(* Logix 5000 project; controller SX_V040001_C001 vendor 1 type 14 code 77 rev 16.23; software revision 16.04; part 25 of 35 *)
(* tags used below, declared in another part *)
   ALL_KINDS : INT[90];
   DRIVE : INT[32];
   Drive_diff_rpm_real : REAL;
   DRIVE_INTERVAL : INT[8];
   Drive_set_prop_rpm_real : REAL;
   EMPTYING : INT[18];
   G_DInput : DINT[3];
   loading : INT[19];
   METERING : INT[44];
   PARAMETER : INT[501];
(* MainProgram, continued *)

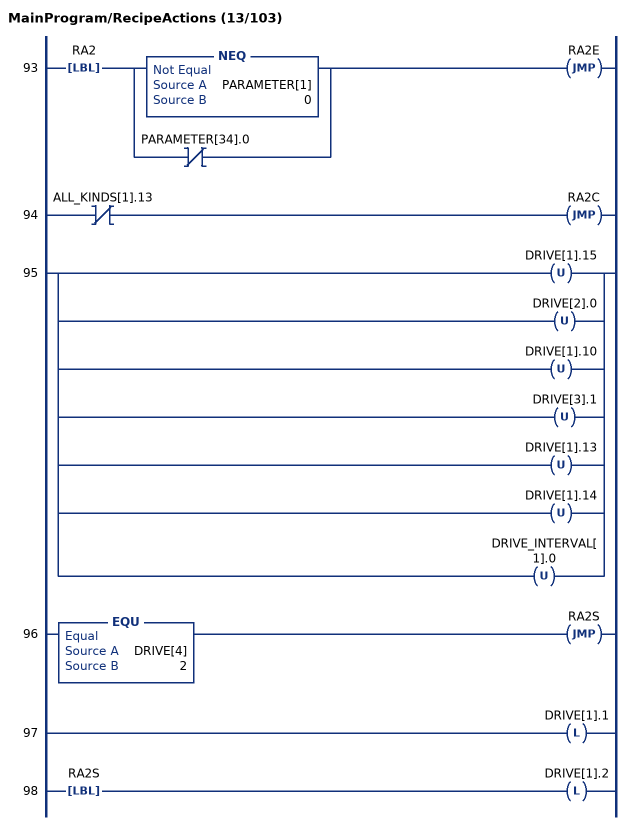
   [picture p547: MainProgram/RecipeActions rungs 93-98]
   93: LBL(RA2)[NEQ(PARAMETER[1],0) ,XIO(PARAMETER[34].0) ]JMP(RA2E);
   94: XIO(ALL_KINDS[1].13)JMP(RA2C);
   95: [OTU(DRIVE[1].15) ,OTU(DRIVE[2].0) ,OTU(DRIVE[1].10) ,OTU(DRIVE[3].1) ,OTU(DRIVE[1].13) ,OTU(DRIVE[1].14) ,OTU(DRIVE_INTERVAL[1].0) ];
   96: EQU(DRIVE[4],2)JMP(RA2S);
   97: OTL(DRIVE[1].1);
   98: LBL(RA2S)OTL(DRIVE[1].2);
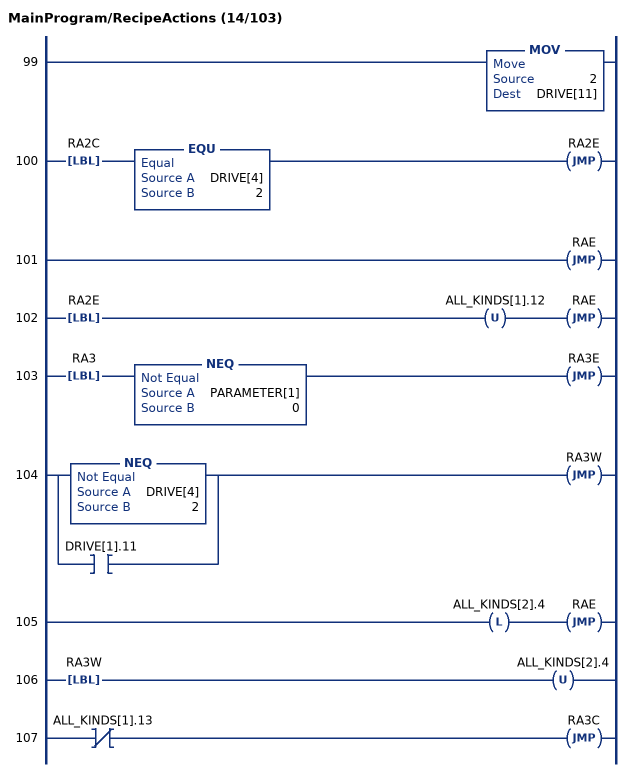
   99: MOV(2,DRIVE[11]);
   100: LBL(RA2C)EQU(DRIVE[4],2)JMP(RA2E);
   101: JMP(RAE);
   102: LBL(RA2E)OTU(ALL_KINDS[1].12)JMP(RAE);
   103: LBL(RA3)NEQ(PARAMETER[1],0)JMP(RA3E);
   104: [NEQ(DRIVE[4],2) ,XIC(DRIVE[1].11) ]JMP(RA3W);
   105: OTL(ALL_KINDS[2].4)JMP(RAE);
   106: LBL(RA3W)OTU(ALL_KINDS[2].4);
   107: XIO(ALL_KINDS[1].13)JMP(RA3C);
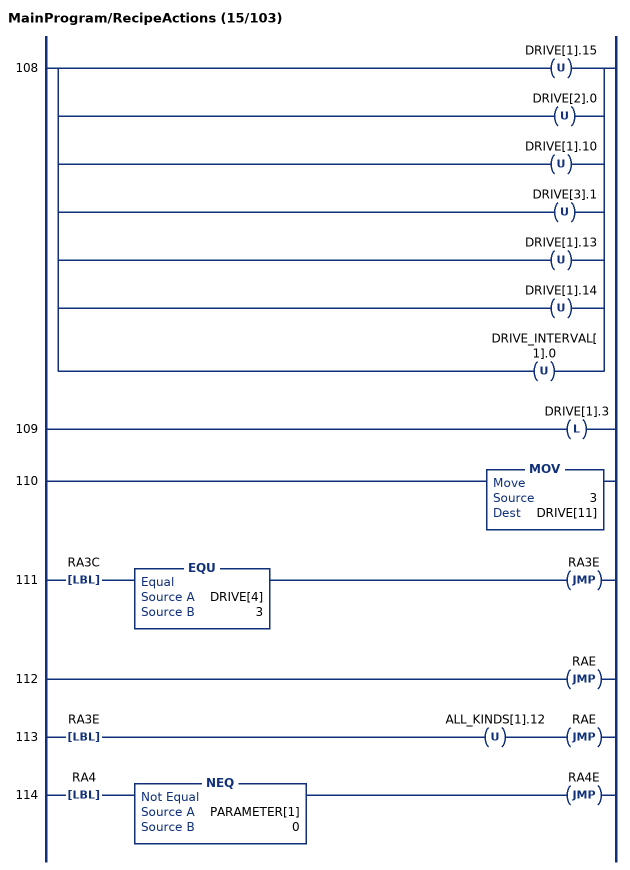
   108: [OTU(DRIVE[1].15) ,OTU(DRIVE[2].0) ,OTU(DRIVE[1].10) ,OTU(DRIVE[3].1) ,OTU(DRIVE[1].13) ,OTU(DRIVE[1].14) ,OTU(DRIVE_INTERVAL[1].0) ];
   109: OTL(DRIVE[1].3);
   110: MOV(3,DRIVE[11]);
   111: LBL(RA3C)EQU(DRIVE[4],3)JMP(RA3E);
   112: JMP(RAE);
   113: LBL(RA3E)OTU(ALL_KINDS[1].12)JMP(RAE);
   114: LBL(RA4)NEQ(PARAMETER[1],0)JMP(RA4E);
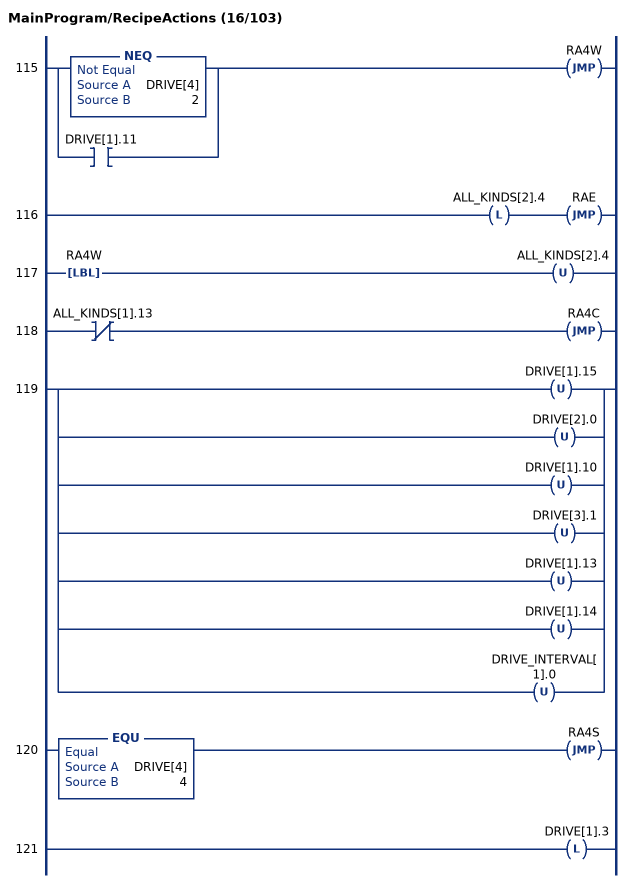
   115: [NEQ(DRIVE[4],2) ,XIC(DRIVE[1].11) ]JMP(RA4W);
   116: OTL(ALL_KINDS[2].4)JMP(RAE);
   117: LBL(RA4W)OTU(ALL_KINDS[2].4);
   118: XIO(ALL_KINDS[1].13)JMP(RA4C);
   119: [OTU(DRIVE[1].15) ,OTU(DRIVE[2].0) ,OTU(DRIVE[1].10) ,OTU(DRIVE[3].1) ,OTU(DRIVE[1].13) ,OTU(DRIVE[1].14) ,OTU(DRIVE_INTERVAL[1].0) ];
   120: EQU(DRIVE[4],4)JMP(RA4S);
   121: OTL(DRIVE[1].3);
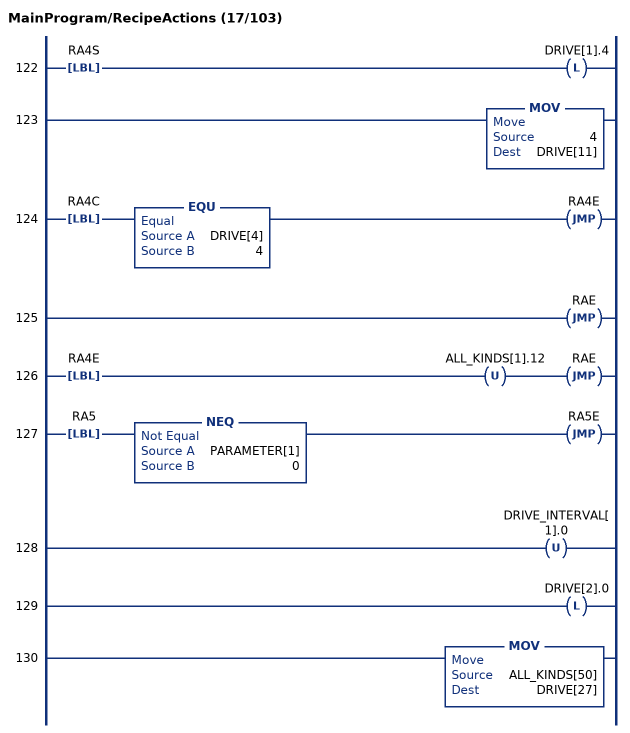
   122: LBL(RA4S)OTL(DRIVE[1].4);
   123: MOV(4,DRIVE[11]);
   124: LBL(RA4C)EQU(DRIVE[4],4)JMP(RA4E);
   125: JMP(RAE);
   126: LBL(RA4E)OTU(ALL_KINDS[1].12)JMP(RAE);
   127: LBL(RA5)NEQ(PARAMETER[1],0)JMP(RA5E);
   128: OTU(DRIVE_INTERVAL[1].0);
   129: OTL(DRIVE[2].0);
   130: MOV(ALL_KINDS[50],DRIVE[27]);
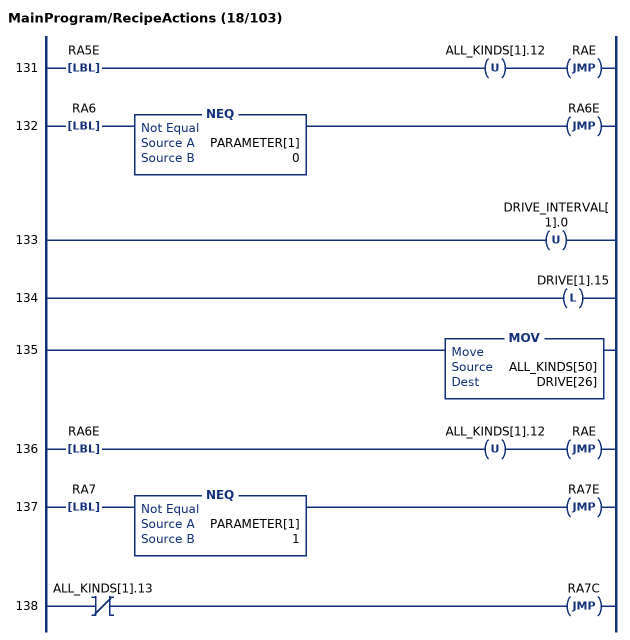
   131: LBL(RA5E)OTU(ALL_KINDS[1].12)JMP(RAE);
   132: LBL(RA6)NEQ(PARAMETER[1],0)JMP(RA6E);
   133: OTU(DRIVE_INTERVAL[1].0);
   134: OTL(DRIVE[1].15);
   135: MOV(ALL_KINDS[50],DRIVE[26]);
   136: LBL(RA6E)OTU(ALL_KINDS[1].12)JMP(RAE);
   137: LBL(RA7)NEQ(PARAMETER[1],1)JMP(RA7E);
   138: XIO(ALL_KINDS[1].13)JMP(RA7C);
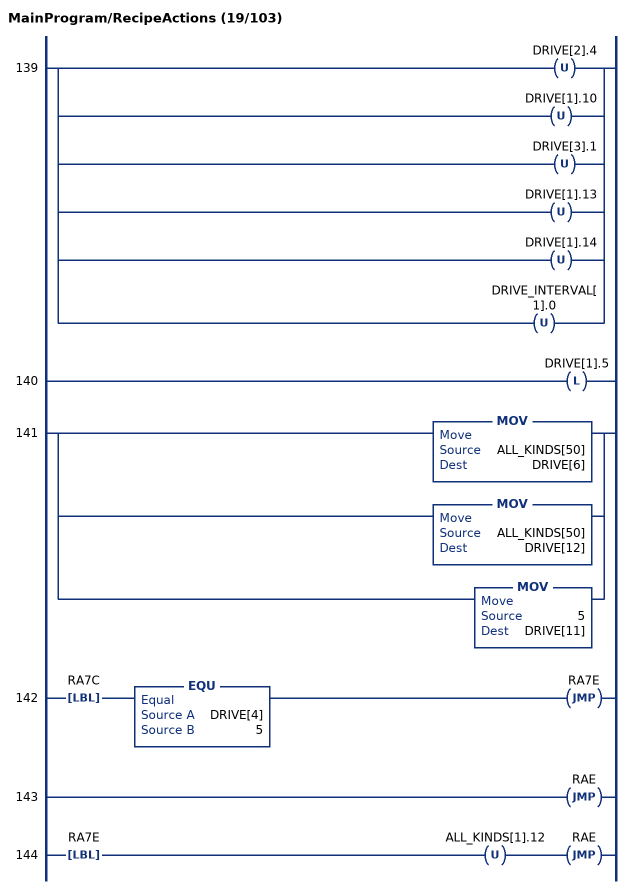
   139: [OTU(DRIVE[2].4) ,OTU(DRIVE[1].10) ,OTU(DRIVE[3].1) ,OTU(DRIVE[1].13) ,OTU(DRIVE[1].14) ,OTU(DRIVE_INTERVAL[1].0) ];
   140: OTL(DRIVE[1].5);
   141: [MOV(ALL_KINDS[50],DRIVE[6]) ,MOV(ALL_KINDS[50],DRIVE[12]) ,MOV(5,DRIVE[11]) ];
   142: LBL(RA7C)EQU(DRIVE[4],5)JMP(RA7E);
   143: JMP(RAE);
   144: LBL(RA7E)OTU(ALL_KINDS[1].12)JMP(RAE);
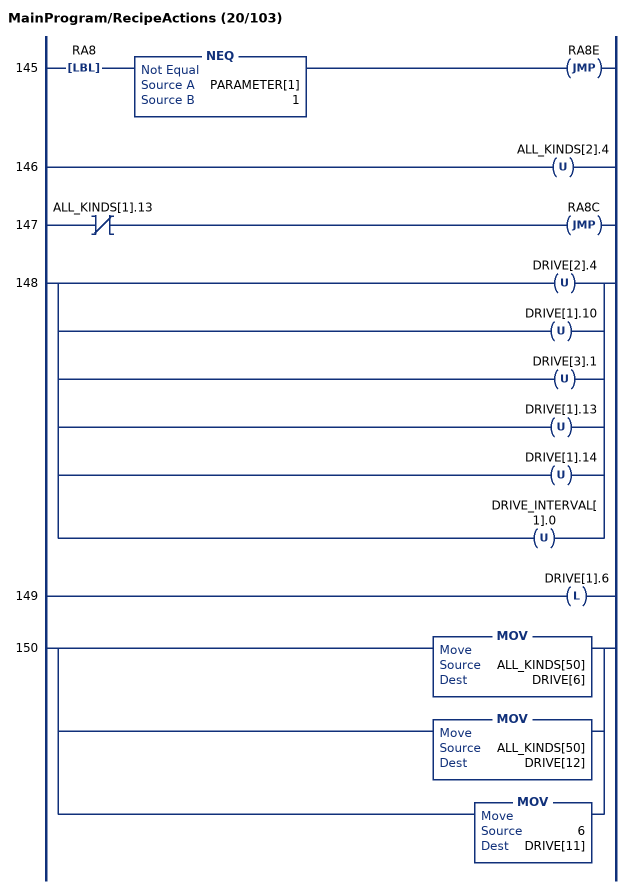
   145: LBL(RA8)NEQ(PARAMETER[1],1)JMP(RA8E);
   146: OTU(ALL_KINDS[2].4);
   147: XIO(ALL_KINDS[1].13)JMP(RA8C);
   148: [OTU(DRIVE[2].4) ,OTU(DRIVE[1].10) ,OTU(DRIVE[3].1) ,OTU(DRIVE[1].13) ,OTU(DRIVE[1].14) ,OTU(DRIVE_INTERVAL[1].0) ];
   149: OTL(DRIVE[1].6);
   150: [MOV(ALL_KINDS[50],DRIVE[6]) ,MOV(ALL_KINDS[50],DRIVE[12]) ,MOV(6,DRIVE[11]) ];
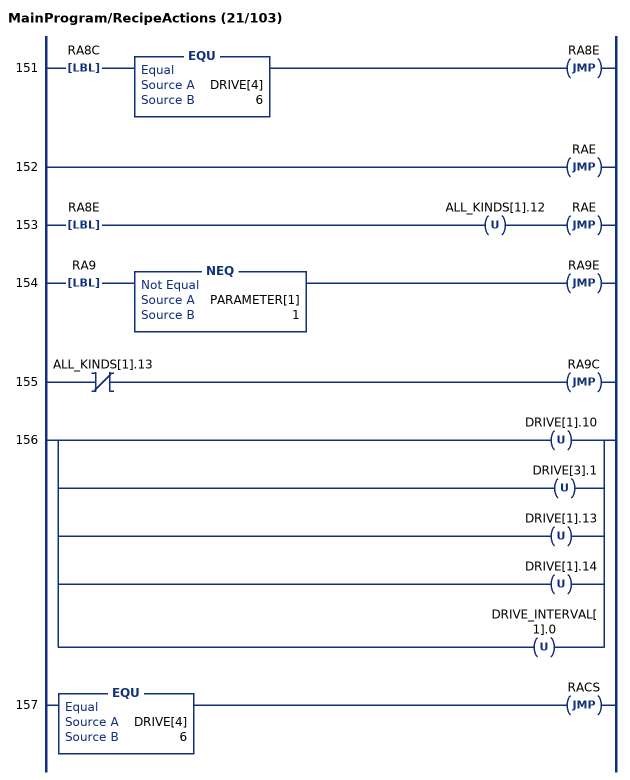
   151: LBL(RA8C)EQU(DRIVE[4],6)JMP(RA8E);
   152: JMP(RAE);
   153: LBL(RA8E)OTU(ALL_KINDS[1].12)JMP(RAE);
   154: LBL(RA9)NEQ(PARAMETER[1],1)JMP(RA9E);
   155: XIO(ALL_KINDS[1].13)JMP(RA9C);
   156: [OTU(DRIVE[1].10) ,OTU(DRIVE[3].1) ,OTU(DRIVE[1].13) ,OTU(DRIVE[1].14) ,OTU(DRIVE_INTERVAL[1].0) ];
   157: EQU(DRIVE[4],6)JMP(RACS);
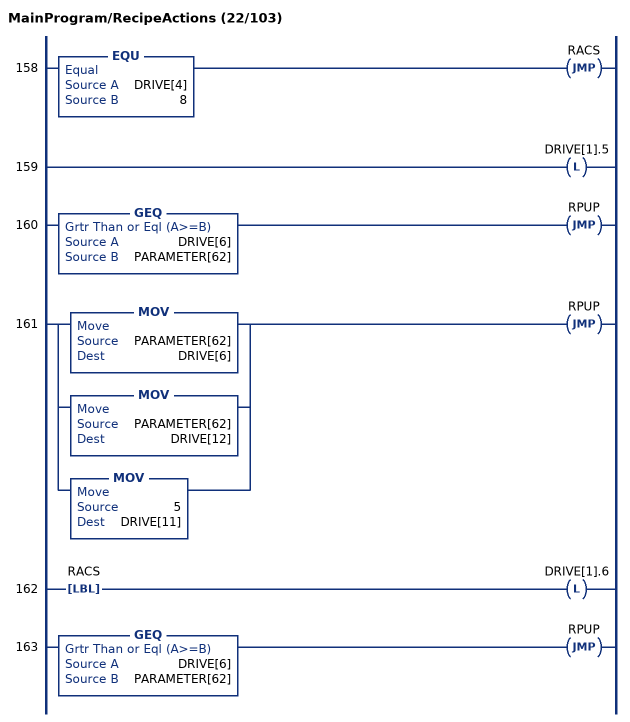
   158: EQU(DRIVE[4],8)JMP(RACS);
   159: OTL(DRIVE[1].5);
   160: GEQ(DRIVE[6],PARAMETER[62])JMP(RPUP);
   161: [MOV(PARAMETER[62],DRIVE[6]) ,MOV(PARAMETER[62],DRIVE[12]) ,MOV(5,DRIVE[11]) ]JMP(RPUP);
   162: LBL(RACS)OTL(DRIVE[1].6);
   163: GEQ(DRIVE[6],PARAMETER[62])JMP(RPUP);
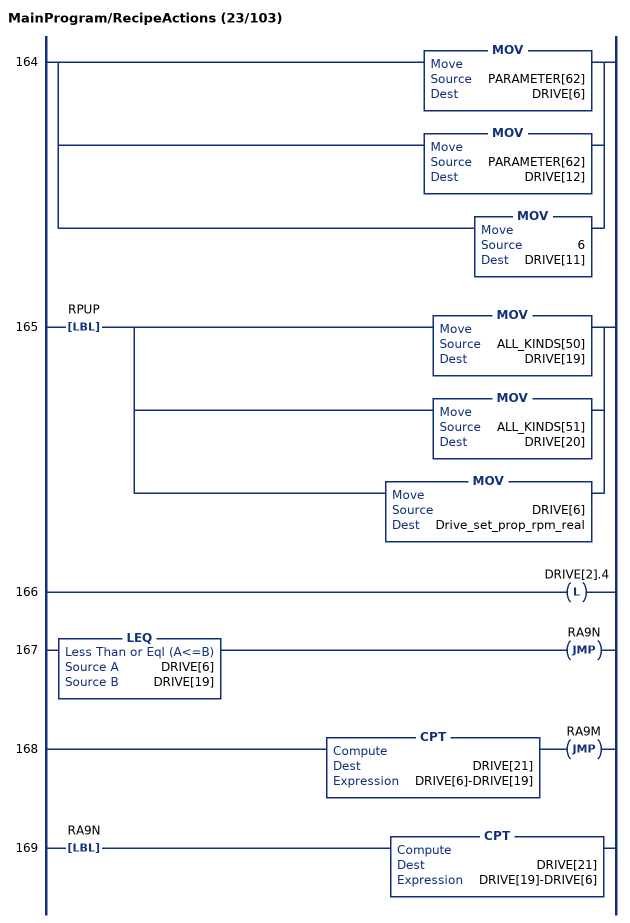
   164: [MOV(PARAMETER[62],DRIVE[6]) ,MOV(PARAMETER[62],DRIVE[12]) ,MOV(6,DRIVE[11]) ];
   165: LBL(RPUP)[MOV(ALL_KINDS[50],DRIVE[19]) ,MOV(ALL_KINDS[51],DRIVE[20]) ,MOV(DRIVE[6],Drive_set_prop_rpm_real) ];
   166: OTL(DRIVE[2].4);
   167: LEQ(DRIVE[6],DRIVE[19])JMP(RA9N);
   168: CPT(DRIVE[21],DRIVE[6]-DRIVE[19])JMP(RA9M);
   169: LBL(RA9N)CPT(DRIVE[21],DRIVE[19]-DRIVE[6]);
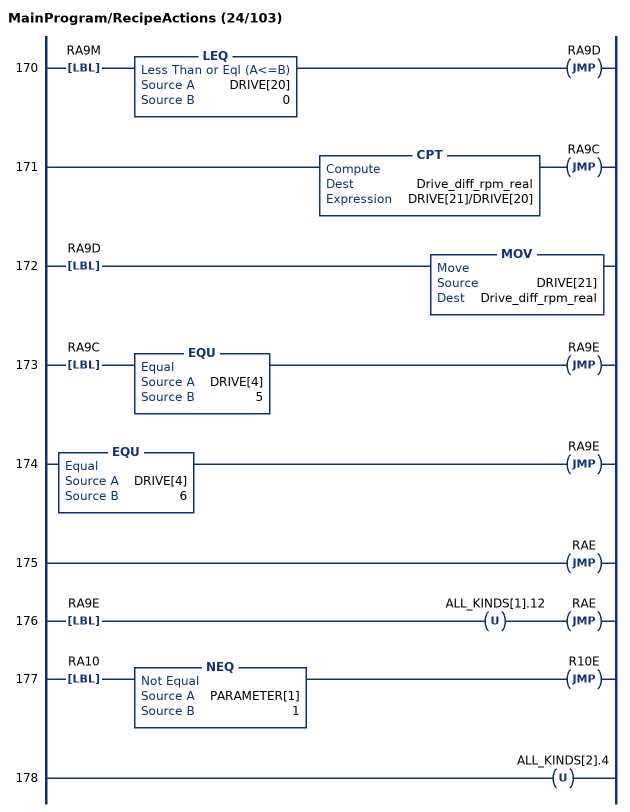
   170: LBL(RA9M)LEQ(DRIVE[20],0)JMP(RA9D);
   171: CPT(Drive_diff_rpm_real,DRIVE[21]/DRIVE[20])JMP(RA9C);
   172: LBL(RA9D)MOV(DRIVE[21],Drive_diff_rpm_real);
   173: LBL(RA9C)EQU(DRIVE[4],5)JMP(RA9E);
   174: EQU(DRIVE[4],6)JMP(RA9E);
   175: JMP(RAE);
   176: LBL(RA9E)OTU(ALL_KINDS[1].12)JMP(RAE);
   177: LBL(RA10)NEQ(PARAMETER[1],1)JMP(R10E);
   178: OTU(ALL_KINDS[2].4);
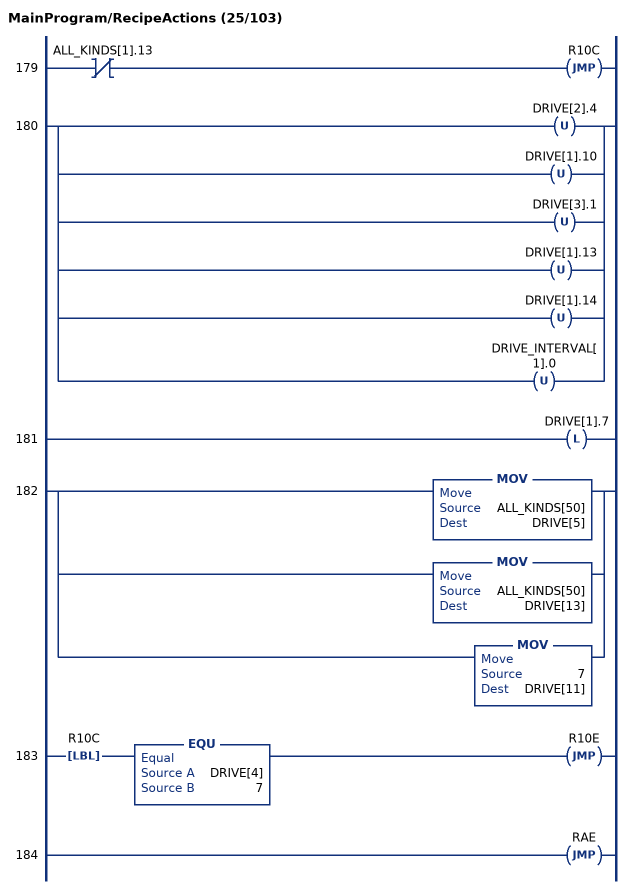
   179: XIO(ALL_KINDS[1].13)JMP(R10C);
   180: [OTU(DRIVE[2].4) ,OTU(DRIVE[1].10) ,OTU(DRIVE[3].1) ,OTU(DRIVE[1].13) ,OTU(DRIVE[1].14) ,OTU(DRIVE_INTERVAL[1].0) ];
   181: OTL(DRIVE[1].7);
   182: [MOV(ALL_KINDS[50],DRIVE[5]) ,MOV(ALL_KINDS[50],DRIVE[13]) ,MOV(7,DRIVE[11]) ];
   183: LBL(R10C)EQU(DRIVE[4],7)JMP(R10E);
   184: JMP(RAE);
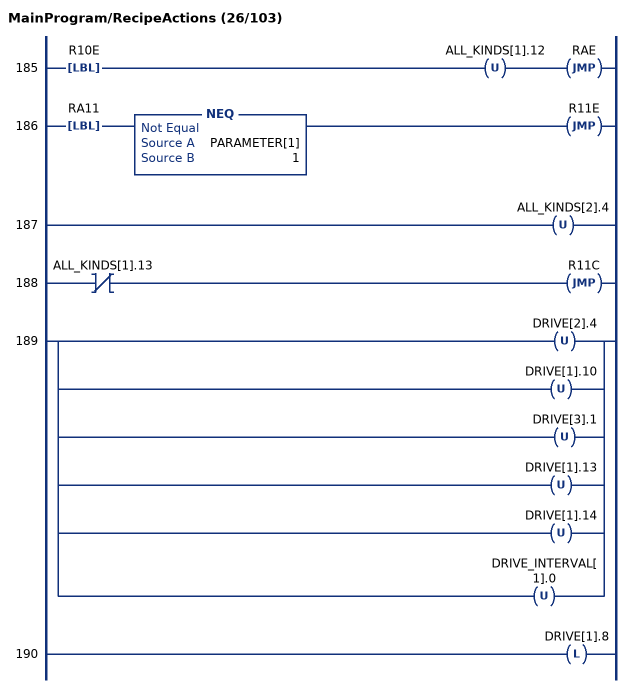
   185: LBL(R10E)OTU(ALL_KINDS[1].12)JMP(RAE);
   186: LBL(RA11)NEQ(PARAMETER[1],1)JMP(R11E);
   187: OTU(ALL_KINDS[2].4);
   188: XIO(ALL_KINDS[1].13)JMP(R11C);
   189: [OTU(DRIVE[2].4) ,OTU(DRIVE[1].10) ,OTU(DRIVE[3].1) ,OTU(DRIVE[1].13) ,OTU(DRIVE[1].14) ,OTU(DRIVE_INTERVAL[1].0) ];
   190: OTL(DRIVE[1].8);
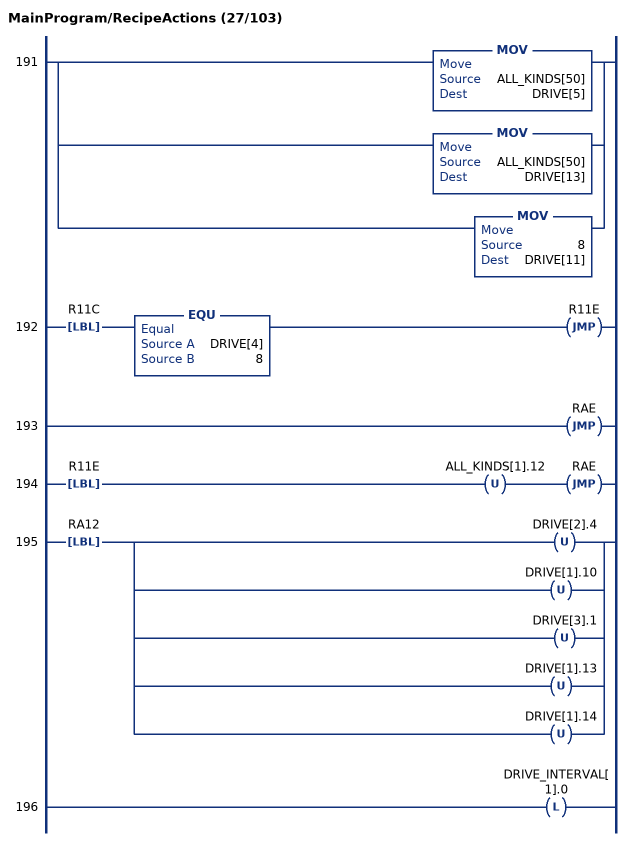
   191: [MOV(ALL_KINDS[50],DRIVE[5]) ,MOV(ALL_KINDS[50],DRIVE[13]) ,MOV(8,DRIVE[11]) ];
   192: LBL(R11C)EQU(DRIVE[4],8)JMP(R11E);
   193: JMP(RAE);
   194: LBL(R11E)OTU(ALL_KINDS[1].12)JMP(RAE);
   195: LBL(RA12)[OTU(DRIVE[2].4) ,OTU(DRIVE[1].10) ,OTU(DRIVE[3].1) ,OTU(DRIVE[1].13) ,OTU(DRIVE[1].14) ];
   196: OTL(DRIVE_INTERVAL[1].0);
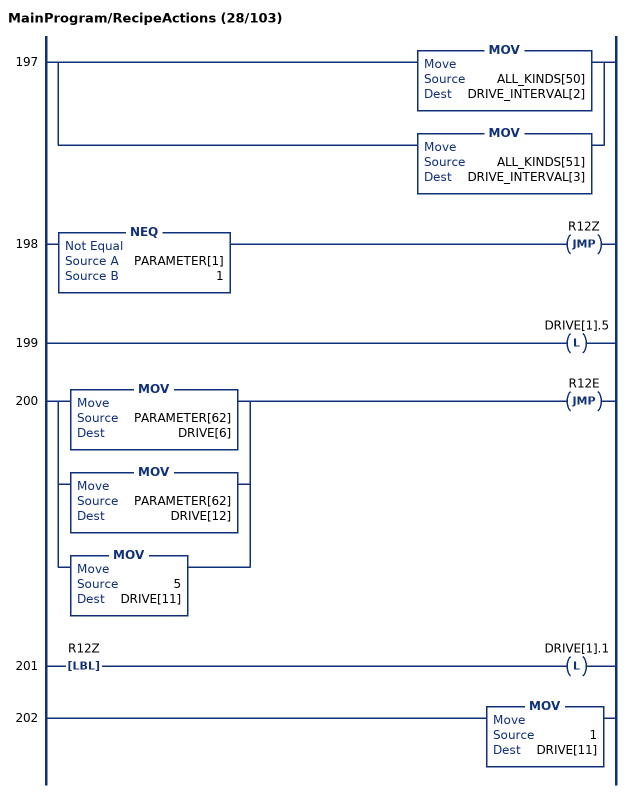
   197: [MOV(ALL_KINDS[50],DRIVE_INTERVAL[2]) ,MOV(ALL_KINDS[51],DRIVE_INTERVAL[3]) ];
   198: NEQ(PARAMETER[1],1)JMP(R12Z);
   199: OTL(DRIVE[1].5);
   200: [MOV(PARAMETER[62],DRIVE[6]) ,MOV(PARAMETER[62],DRIVE[12]) ,MOV(5,DRIVE[11]) ]JMP(R12E);
   201: LBL(R12Z)OTL(DRIVE[1].1);
   202: MOV(1,DRIVE[11]);
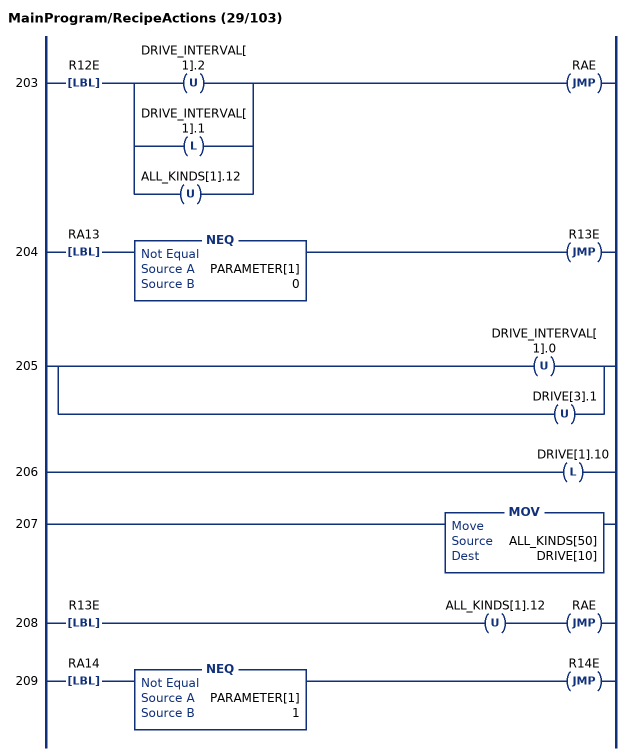
   203: LBL(R12E)[OTU(DRIVE_INTERVAL[1].2) ,OTL(DRIVE_INTERVAL[1].1) ,OTU(ALL_KINDS[1].12) ]JMP(RAE);
   204: LBL(RA13)NEQ(PARAMETER[1],0)JMP(R13E);
   205: [OTU(DRIVE_INTERVAL[1].0) ,OTU(DRIVE[3].1) ];
   206: OTL(DRIVE[1].10);
   207: MOV(ALL_KINDS[50],DRIVE[10]);
   208: LBL(R13E)OTU(ALL_KINDS[1].12)JMP(RAE);
   209: LBL(RA14)NEQ(PARAMETER[1],1)JMP(R14E);
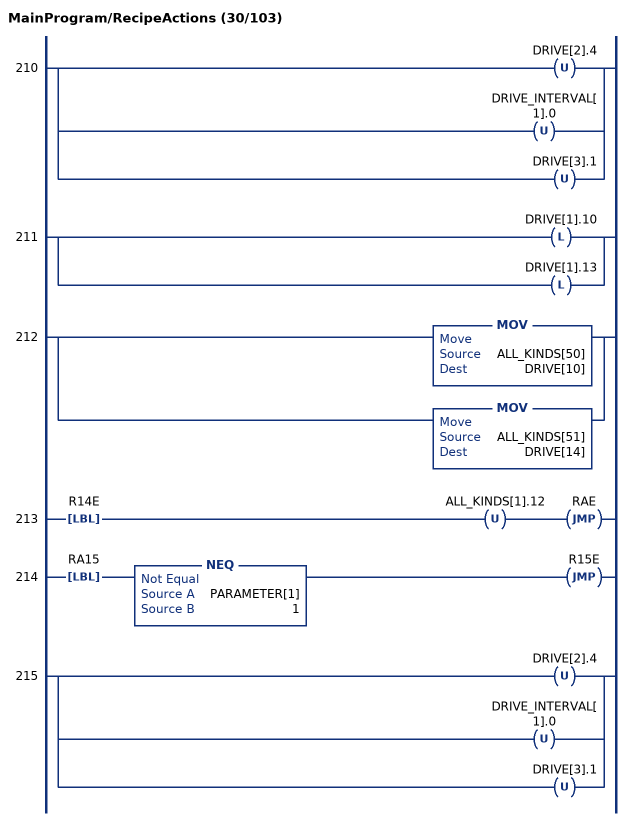
   210: [OTU(DRIVE[2].4) ,OTU(DRIVE_INTERVAL[1].0) ,OTU(DRIVE[3].1) ];
   211: [OTL(DRIVE[1].10) ,OTL(DRIVE[1].13) ];
   212: [MOV(ALL_KINDS[50],DRIVE[10]) ,MOV(ALL_KINDS[51],DRIVE[14]) ];
   213: LBL(R14E)OTU(ALL_KINDS[1].12)JMP(RAE);
   214: LBL(RA15)NEQ(PARAMETER[1],1)JMP(R15E);
   215: [OTU(DRIVE[2].4) ,OTU(DRIVE_INTERVAL[1].0) ,OTU(DRIVE[3].1) ];
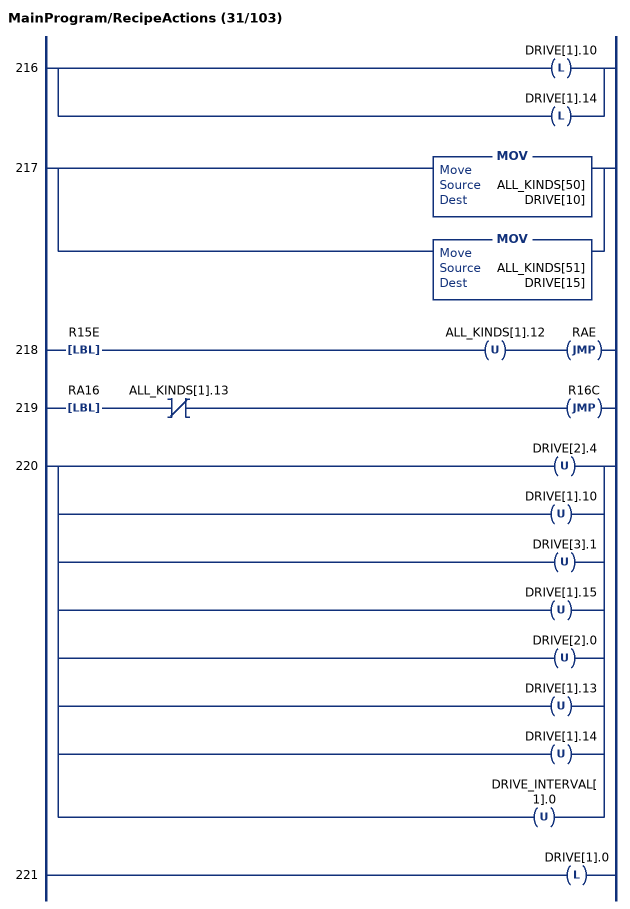
   216: [OTL(DRIVE[1].10) ,OTL(DRIVE[1].14) ];
   217: [MOV(ALL_KINDS[50],DRIVE[10]) ,MOV(ALL_KINDS[51],DRIVE[15]) ];
   218: LBL(R15E)OTU(ALL_KINDS[1].12)JMP(RAE);
   219: LBL(RA16)XIO(ALL_KINDS[1].13)JMP(R16C);
   220: [OTU(DRIVE[2].4) ,OTU(DRIVE[1].10) ,OTU(DRIVE[3].1) ,OTU(DRIVE[1].15) ,OTU(DRIVE[2].0) ,OTU(DRIVE[1].13) ,OTU(DRIVE[1].14) ,OTU(DRIVE_INTERVAL[1].0) ];
   221: OTL(DRIVE[1].0);
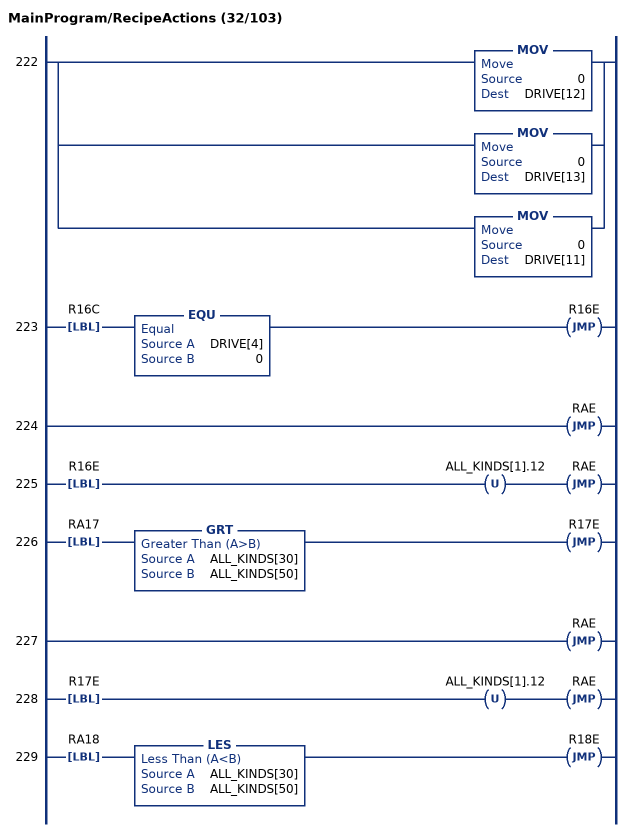
   222: [MOV(0,DRIVE[12]) ,MOV(0,DRIVE[13]) ,MOV(0,DRIVE[11]) ];
   223: LBL(R16C)EQU(DRIVE[4],0)JMP(R16E);
   224: JMP(RAE);
   225: LBL(R16E)OTU(ALL_KINDS[1].12)JMP(RAE);
   226: LBL(RA17)GRT(ALL_KINDS[30],ALL_KINDS[50])JMP(R17E);
   227: JMP(RAE);
   228: LBL(R17E)OTU(ALL_KINDS[1].12)JMP(RAE);
   229: LBL(RA18)LES(ALL_KINDS[30],ALL_KINDS[50])JMP(R18E);
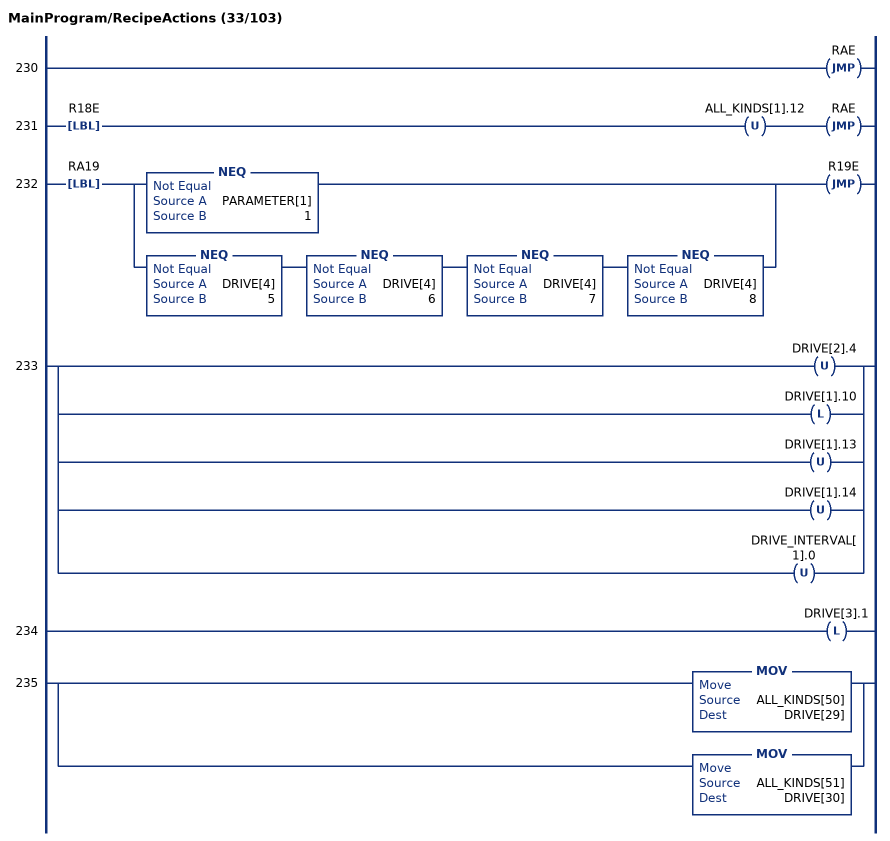
   230: JMP(RAE);
   231: LBL(R18E)OTU(ALL_KINDS[1].12)JMP(RAE);
   232: LBL(RA19)[NEQ(PARAMETER[1],1) ,NEQ(DRIVE[4],5) NEQ(DRIVE[4],6) NEQ(DRIVE[4],7) NEQ(DRIVE[4],8) ]JMP(R19E);
   233: [OTU(DRIVE[2].4) ,OTL(DRIVE[1].10) ,OTU(DRIVE[1].13) ,OTU(DRIVE[1].14) ,OTU(DRIVE_INTERVAL[1].0) ];
   234: OTL(DRIVE[3].1);
   235: [MOV(ALL_KINDS[50],DRIVE[29]) ,MOV(ALL_KINDS[51],DRIVE[30]) ];
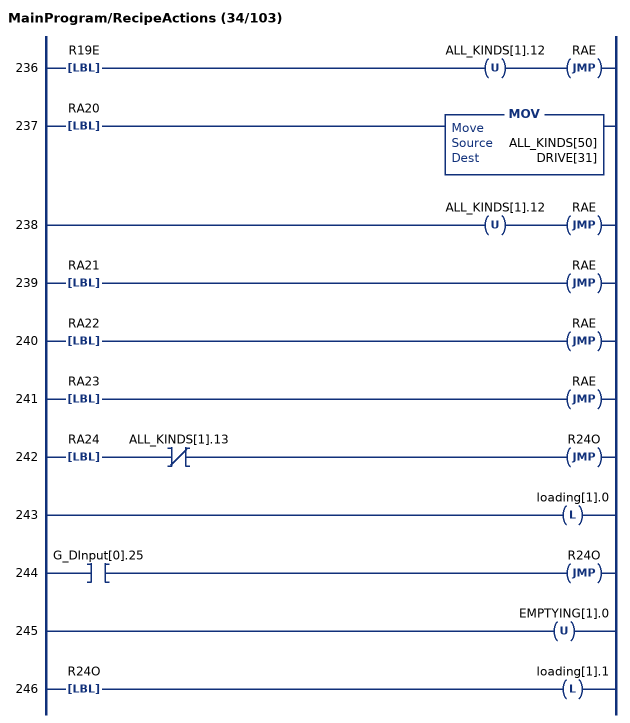
   236: LBL(R19E)OTU(ALL_KINDS[1].12)JMP(RAE);
   237: LBL(RA20)MOV(ALL_KINDS[50],DRIVE[31]);
   238: OTU(ALL_KINDS[1].12)JMP(RAE);
   239: LBL(RA21)JMP(RAE);
   240: LBL(RA22)JMP(RAE);
   241: LBL(RA23)JMP(RAE);
   242: LBL(RA24)XIO(ALL_KINDS[1].13)JMP(R24O);
   243: OTL(loading[1].0);
   244: XIC(G_DInput[0].25)JMP(R24O);
   245: OTU(EMPTYING[1].0);
   246: LBL(R24O)OTL(loading[1].1);
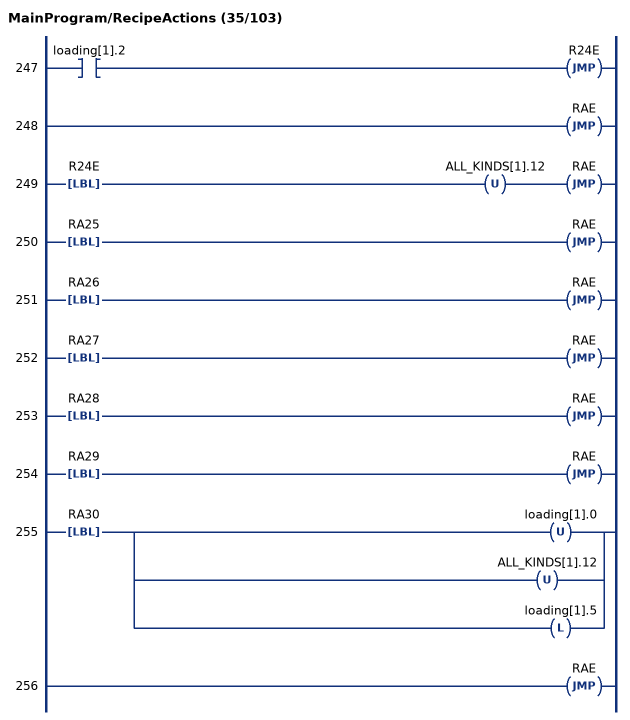
   247: XIC(loading[1].2)JMP(R24E);
   248: JMP(RAE);
   249: LBL(R24E)OTU(ALL_KINDS[1].12)JMP(RAE);
   250: LBL(RA25)JMP(RAE);
   251: LBL(RA26)JMP(RAE);
   252: LBL(RA27)JMP(RAE);
   253: LBL(RA28)JMP(RAE);
   254: LBL(RA29)JMP(RAE);
   255: LBL(RA30)[OTU(loading[1].0) ,OTU(ALL_KINDS[1].12) ,OTL(loading[1].5) ];
   256: JMP(RAE);
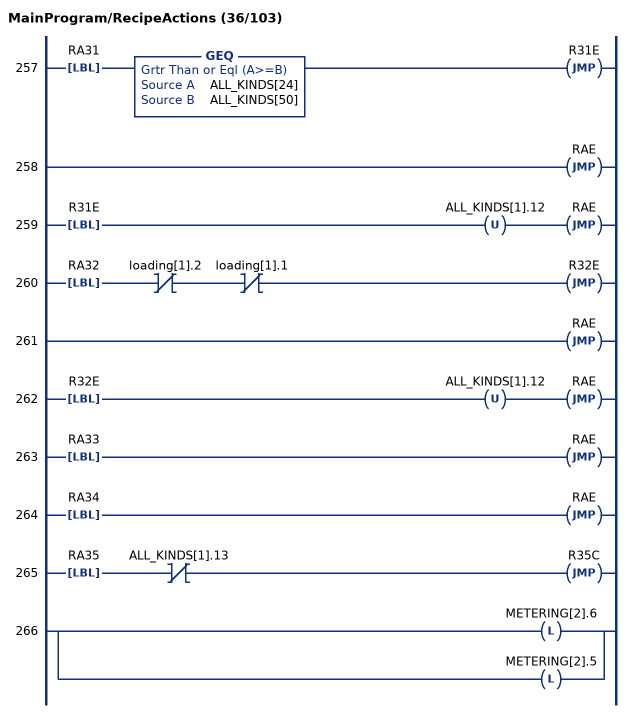
   257: LBL(RA31)GEQ(ALL_KINDS[24],ALL_KINDS[50])JMP(R31E);
   258: JMP(RAE);
   259: LBL(R31E)OTU(ALL_KINDS[1].12)JMP(RAE);
   260: LBL(RA32)XIO(loading[1].2)XIO(loading[1].1)JMP(R32E);
   261: JMP(RAE);
   262: LBL(R32E)OTU(ALL_KINDS[1].12)JMP(RAE);
   263: LBL(RA33)JMP(RAE);
   264: LBL(RA34)JMP(RAE);
   265: LBL(RA35)XIO(ALL_KINDS[1].13)JMP(R35C);
   266: [OTL(METERING[2].6) ,OTL(METERING[2].5) ];
